{attribute 'strict'}
{attribute 'to_string'}
TYPE eProgress :
(
	INIT := 0,
	ACKNOWLEDGE := 1,
	RUNNING := 2,
	FINALIZED := 3,
	ABORTED := 4
);
END_TYPE

(* stored: Version 1.1.0.1, ProductVersion 3.1.4026.18
   DUT eProgress: Id {d1a825b7-0b16-4bfe-bb2c-8862a9623c51} *)
